(* IEC 61131-3 sources: POMIRTS_lab3/AS/Library_2/AsNxPnS, 3 files *)

(* ---- AsNxPnS.typ ---- *)
TYPE
	PnSoftwareRevisionType : 	STRUCT
		Prefix : USINT;
		X : USINT;
		Y : USINT;
		Z : USINT;
	END_STRUCT;
	PnIm0Type : 	STRUCT
		VendorID : UINT;
		OrderID : ARRAY[0..19]OF USINT;
		SerialNumber : ARRAY[0..15]OF USINT;
		HardwareRevision : UINT;
		SoftwareRevision : PnSoftwareRevisionType;
		RevisionCounter : UINT;
		ProfileID : UINT;
		ProfileSpecificType : UINT;
		IMVersion : UINT;
		IMSupported : UINT;
	END_STRUCT;
	PnIm5Type : 	STRUCT
		Annotation : ARRAY[0..63]OF USINT;
		OrderID : ARRAY[0..63]OF USINT;
		VendorID : UINT;
		SerialNumber : ARRAY[0..15]OF USINT;
		HardwareRevision : UINT;
		SoftwareRevision : PnSoftwareRevisionType;
	END_STRUCT;
END_TYPE

(* ---- AsNxPnS.fun ---- *)
{REDUND_CONTEXT} {REDUND_UNREPLICABLE} FUNCTION_BLOCK nxpnsProcessAlarm		(*process alarm*)
	VAR_INPUT
		enable			: BOOL;			(*enables execution*)
		pDevice			: UDINT;		(*interface name given as a pointer, e.g., "SL<x>.SS<y>.IF<z>"*)
		deviceHandle	: UDINT;		(*profinet slave handle*)
		alarmHandle		: UDINT;		(*alarm handle*)
		userStructId	: UINT;			(*user structure identifier*)
		api				: UDINT;		(*api*)
		slot			: UDINT;		(*slot*)
		subslot			: UDINT;		(*subslot*)
		alarmDataLen	: UINT;			(*alarm data length*)
		pAlarmData		: UDINT;		(*alarm data given as pointer*)
	END_VAR
	VAR
        _state			: UINT;			(*internal variable*)
		_result			: UINT;			(*internal variable*)
        _srcId			: UDINT;		(*internal variable*)
	END_VAR
	VAR_OUTPUT
		status			: UINT;			(*execution status: ERR_OK, ERR_FUB_ENABLE_FALSE, ERR_FUB_BUSY, 0xXXXX = see help*)
		pnStatus		: UDINT;		(*profinet stack status*)
		pnIoStatus		: UDINT;		(*profinet io status*)
	END_VAR
END_FUNCTION_BLOCK

{REDUND_CONTEXT} {REDUND_UNREPLICABLE} FUNCTION_BLOCK nxpnsDiagnosisAlarm		(*diagnosis alarm*)
	VAR_INPUT
		enable			: BOOL;			(*enables execution*)
		pDevice			: UDINT;		(*interface name given as a pointer, e.g., "SL<x>.SS<y>.IF<z>"*)
		deviceHandle	: UDINT;		(*profinet slave handle*)
		alarmHandle		: UDINT;		(*alarm handle*)
		diagHandle		: UDINT;		(*diagnosis handle*)
	END_VAR
	VAR
        _state			: UINT;			(*internal variable*)
		_result			: UINT;			(*internal variable*)
        _srcId			: UDINT;		(*internal variable*)
	END_VAR
	VAR_OUTPUT
		status			: UINT;			(*execution status: ERR_OK, ERR_FUB_ENABLE_FALSE, ERR_FUB_BUSY, 0xXXXX = see help*)
		pnStatus		: UDINT;		(*profinet stack status*)
		pnIoStatus		: UDINT;		(*profinet io status*)
	END_VAR
END_FUNCTION_BLOCK

{REDUND_CONTEXT} {REDUND_UNREPLICABLE} FUNCTION_BLOCK nxpnsPlugModule			(*plug module*)
	VAR_INPUT
		enable			: BOOL;			(*enables execution*)
		pDevice			: UDINT;		(*interface name given as a pointer, e.g., "SL<x>.SS<y>.IF<z>"*)
		deviceHandle	: UDINT;		(*profinet slave handle*)
		api				: UDINT;		(*api*)
		slot			: UDINT;		(*slot*)
		moduleId		: UDINT;		(*module identifier*)
		moduleState		: UINT;			(*module state*)
	END_VAR
	VAR
        _state			: UINT;			(*internal variable*)
		_result			: UINT;			(*internal variable*)
        _srcId			: UDINT;		(*internal variable*)
	END_VAR
	VAR_OUTPUT
		status			: UINT;			(*execution status: ERR_OK, ERR_FUB_ENABLE_FALSE, ERR_FUB_BUSY, 0xXXXX = see help*)
		pnStatus		: UDINT;		(*profinet stack status*)
	END_VAR
END_FUNCTION_BLOCK

{REDUND_CONTEXT} {REDUND_UNREPLICABLE} FUNCTION_BLOCK nxpnsPullModule			(*pull module*)
	VAR_INPUT
		enable			: BOOL;			(*enables execution*)
		pDevice			: UDINT;		(*interface name given as a pointer, e.g., "SL<x>.SS<y>.IF<z>"*)
		deviceHandle	: UDINT;		(*profinet slave handle*)
		api				: UDINT;		(*api*)
		slot			: UDINT;		(*slot*)
	END_VAR
	VAR
        _state			: UINT;			(*internal variable*)
		_result			: UINT;			(*internal variable*)
        _srcId			: UDINT;		(*internal variable*)
	END_VAR
	VAR_OUTPUT
		status			: UINT;			(*execution status: ERR_OK, ERR_FUB_ENABLE_FALSE, ERR_FUB_BUSY, 0xXXXX = see help*)
		pnStatus		: UDINT;		(*profinet stack status*)
	END_VAR
END_FUNCTION_BLOCK

{REDUND_CONTEXT} {REDUND_UNREPLICABLE} FUNCTION_BLOCK nxpnsGetHandle			(*get slave handle*)
	VAR_INPUT
		enable			: BOOL;			(*enables execution*)
		pDevice			: UDINT;		(*interface name given as a pointer, e.g., "SL<x>.SS<y>.IF<z>"*)
	END_VAR
	VAR
        _state			: UINT;			(*internal variable*)
		_result			: UINT;			(*internal variable*)
        _srcId			: UDINT;		(*internal variable*)
	END_VAR
	VAR_OUTPUT
		status			: UINT;			(*execution status: ERR_OK, ERR_FUB_ENABLE_FALSE, ERR_FUB_BUSY, 0xXXXX = see help*)
		pnStatus		: UDINT;		(*profinet stack status*)
		deviceHandle	: UDINT;		(*profinet slave handle*)
	END_VAR
END_FUNCTION_BLOCK

{REDUND_CONTEXT} {REDUND_UNREPLICABLE} FUNCTION_BLOCK nxpnsAddChannelDiag		(*add channel diagnosis*)
	VAR_INPUT
		enable			: BOOL;			(*enables execution*)
		pDevice			: UDINT;		(*interface name given as a pointer, e.g., "SL<x>.SS<y>.IF<z>"*)
		api				: UDINT;		(*api*)
		slot			: UDINT;		(*slot*)
		subslot			: UDINT;		(*subslot*)
		channelNum		: UINT;			(*channel number*)
		channelProp		: UINT;			(*channel property*)
		channelErrType	: UINT;			(*channel error type*)
	END_VAR
	VAR
        _state			: UINT;			(*internal variable*)
		_result			: UINT;			(*internal variable*)
        _srcId			: UDINT;		(*internal variable*)
	END_VAR
	VAR_OUTPUT
		status			: UINT;			(*execution status: ERR_OK, ERR_FUB_ENABLE_FALSE, ERR_FUB_BUSY, 0xXXXX = see help*)
		pnStatus		: UDINT;		(*profinet stack status*)
		diagHandle		: UDINT;		(*profinet diagnosis handle*)
	END_VAR
END_FUNCTION_BLOCK

{REDUND_CONTEXT} {REDUND_UNREPLICABLE} FUNCTION_BLOCK nxpnsAddExtChannelDiag	(*add channel diagnosis*)
	VAR_INPUT
		enable			: BOOL;			(*enables execution*)
		pDevice			: UDINT;		(*interface name given as a pointer, e.g., "SL<x>.SS<y>.IF<z>"*)
		api				: UDINT;		(*api*)
		slot			: UDINT;		(*slot*)
		subslot			: UDINT;		(*subslot*)
		channelNum		: UINT;			(*channel number*)
		channelProp		: UINT;			(*channel property*)
		channelErrType	: UINT;			(*channel error type*)
		extChannelAddValue	: UDINT;	(*reserved for future use, set to zero*)
		extChannelErrType	: UINT;		(*extended channel error type*)
	END_VAR
	VAR
        _state			: UINT;			(*internal variable*)
		_result			: UINT;			(*internal variable*)
        _srcId			: UDINT;		(*internal variable*)
	END_VAR
	VAR_OUTPUT
		status			: UINT;			(*execution status: ERR_OK, ERR_FUB_ENABLE_FALSE, ERR_FUB_BUSY, 0xXXXX = see help*)
		pnStatus		: UDINT;		(*profinet stack status*)
		diagHandle		: UDINT;		(*profinet diagnosis handle*)
	END_VAR
END_FUNCTION_BLOCK

{REDUND_CONTEXT} {REDUND_UNREPLICABLE} FUNCTION_BLOCK nxpnsAddGenChannelDiag	(*add channel diagnosis*)
	VAR_INPUT
		enable			: BOOL;			(*enables execution*)
		pDevice			: UDINT;		(*interface name given as a pointer, e.g., "SL<x>.SS<y>.IF<z>"*)
		api				: UDINT;		(*api*)
		slot			: UDINT;		(*slot*)
		subslot			: UDINT;		(*subslot*)
		channelNum		: UINT;			(*channel number*)
		channelProp		: UINT;			(*channel property*)
		channelErrType	: UINT;			(*channel error type*)
		userStructId	: UINT;			(*user structure identifier*)
		diagDataLen		: UINT;			(*diagnosis data length*)
		pDiagData		: UDINT;		(*diagnosis data given as pointer*)
	END_VAR
	VAR
        _state			: UINT;			(*internal variable*)
		_result			: UINT;			(*internal variable*)
        _srcId			: UDINT;		(*internal variable*)
	END_VAR
	VAR_OUTPUT
		status			: UINT;			(*execution status: ERR_OK, ERR_FUB_ENABLE_FALSE, ERR_FUB_BUSY, 0xXXXX = see help*)
		pnStatus		: UDINT;		(*profinet stack status*)
		diagHandle		: UDINT;		(*profinet diagnosis handle*)
	END_VAR
END_FUNCTION_BLOCK

{REDUND_CONTEXT} {REDUND_UNREPLICABLE} FUNCTION_BLOCK nxpnsRemChannelDiag		(*remove channel diagnosis*)
	VAR_INPUT
		enable			: BOOL;			(*enables execution*)
		pDevice			: UDINT;		(*interface name given as a pointer, e.g., "SL<x>.SS<y>.IF<z>"*)
		diagHandle		: UDINT;		(*diagnosis handle*)
	END_VAR
	VAR
        _state			: UINT;			(*internal variable*)
		_result			: UINT;			(*internal variable*)
        _srcId			: UDINT;		(*internal variable*)
	END_VAR
	VAR_OUTPUT
		status			: UINT;			(*execution status: ERR_OK, ERR_FUB_ENABLE_FALSE, ERR_FUB_BUSY, 0xXXXX = see help*)
		pnStatus		: UDINT;		(*profinet stack status*)
	END_VAR
END_FUNCTION_BLOCK

{REDUND_CONTEXT} {REDUND_UNREPLICABLE} FUNCTION_BLOCK nxpnsSetName				(*set station name*)
	VAR_INPUT
		enable			: BOOL;			(*enables execution*)
		pDevice			: UDINT;		(*interface name given as a pointer, e.g., "SL<x>.SS<y>.IF<z>"*)
		pName			: UDINT;		(*new station name*)
	END_VAR
	VAR
        _state			: UINT;			(*internal variable*)
		_result			: UINT;			(*internal variable*)
        _srcId			: UDINT;		(*internal variable*)
	END_VAR
	VAR_OUTPUT
		status			: UINT;			(*execution status: ERR_OK, ERR_FUB_ENABLE_FALSE, ERR_FUB_BUSY, 0xXXXX = see help*)
		pnStatus		: UDINT;		(*profinet stack status*)
	END_VAR
END_FUNCTION_BLOCK

{REDUND_CONTEXT} {REDUND_UNREPLICABLE} FUNCTION_BLOCK nxpnsStartBusComm		(*start bus communication*)
	VAR_INPUT
		enable			: BOOL;			(*enables execution*)
		pDevice			: UDINT;		(*interface name given as a pointer, e.g., "SL<x>.SS<y>.IF<z>"*)
	END_VAR
	VAR
        _state			: UINT;			(*internal variable*)
		_result			: UINT;			(*internal variable*)
        _srcId			: UDINT;		(*internal variable*)
	END_VAR
	VAR_OUTPUT
		status			: UINT;			(*execution status: ERR_OK, ERR_FUB_ENABLE_FALSE, ERR_FUB_BUSY, 0xXXXX = see help*)
		pnStatus		: UDINT;		(*profinet stack status*)
	END_VAR
END_FUNCTION_BLOCK

{REDUND_CONTEXT} {REDUND_UNREPLICABLE} FUNCTION_BLOCK nxpnsGetIm0 (*Gets the I&M0 data set for this device*)
	VAR_INPUT
		enable		: BOOL;				(*Enables execution.*)
		pDevice		: UDINT;			(*Name of the profinet device e.g. SS1.IF1.*)
	END_VAR
	VAR_OUTPUT
		status		: DINT;  			(*Status information.*)
		pnStatus	: UDINT;			(*Profinet stack status*)
		IM0 		: PnIm0Type;		(*I&M0 data*)
	END_VAR
	VAR
		_state		: UINT;				(*internal variable*)
		_result		: UINT;				(*internal variable*)
        _srcId		: UDINT;			(*internal variable*)
	END_VAR
END_FUNCTION_BLOCK

{REDUND_CONTEXT} {REDUND_UNREPLICABLE} FUNCTION_BLOCK nxpnsSetOem (*Sets the OEM data for this device*)
	VAR_INPUT
		enable		: BOOL;				(*Enables execution.*)
		pDevice		: UDINT;			(*Name of the profinet device e.g. SS1.IF1.*)
		DeviceID	: UINT;				(*Profinet Device Identification*)
		DeviceType	: ARRAY[0..24]OF USINT; (*Profinet Device Type*)
		IM0 		: PnIm0Type;		(*I&M0 data to be set*)
	END_VAR
	VAR_OUTPUT
		status		: DINT;  			(*Status information.*)
		pnStatus	: UDINT;			(*Profinet stack status*)
	END_VAR
	VAR
		_state		: UINT;				(*internal variable*)
		_result		: UINT;				(*internal variable*)
        _srcId		: UDINT;			(*internal variable*)
	END_VAR
END_FUNCTION_BLOCK

{REDUND_CONTEXT} {REDUND_UNREPLICABLE} FUNCTION_BLOCK nxpnsSetIm5 (*Sets the I&M5 data for this device*)
	VAR_INPUT
		enable		: BOOL;				(*Enables execution.*)
		pDevice		: UDINT;			(*Name of the profinet device e.g. SS1.IF1.*)
		IM5 		: PnIm5Type;		(*I&M5 data to be set*)
	END_VAR
	VAR_OUTPUT
		status		: DINT;  			(*Status information.*)
		pnStatus	: UDINT;			(*Profinet stack status*)
	END_VAR
	VAR
		_state		: UINT;				(*internal variable*)
		_result		: UINT;				(*internal variable*)
        _srcId		: UDINT;			(*internal variable*)
	END_VAR
END_FUNCTION_BLOCK

(* ---- AsNxPnS.var ---- *)
VAR CONSTANT
	nxpnsERR_INVALID_DEVICE				: UINT	:= 35320;		(*error invalid device*)
	nxpnsERR_SEND_MESSAGE				: UINT	:= 35321;		(*error send message*)
	nxpnsERR_TIMEOUT					: UINT	:= 35322;		(*error timeout*)
	nxpnsERR_PROFINET_STACK				: UINT	:= 35323;		(*error receive message*)
	nxpnsERR_PARAMETER					: UINT	:= 35324;		(*error invalid parameter*)

	nxpnsMOD_PLUG_CORRECT_MOD			: UINT	:= 16#0000;		(*plug correct module*)
	nxpnsMOD_PLUG_SUBSTITUTE_MOD		: UINT	:= 16#0001;		(*plug substitute module*)

	nxpnsALARM_DATALEN_MAX				: UDINT	:= 1024;		(*max alarm data length*)

	nxpnsCERR_SHORT_CIRCUIT				: UINT	:= 16#0001;		(*channel error type short circuit*)
	nxpnsCERR_UNDERVOLTAGE				: UINT	:= 16#0002;		(*channel error type undervoltaqe*)
	nxpnsCERR_OVERVOLTAGE				: UINT	:= 16#0003;		(*channel error type overvoltage*)
	nxpnsCERR_OVERLOAD					: UINT	:= 16#0004;		(*channel error type overload*)
	nxpnsCERR_OVERTEMPERATURE			: UINT	:= 16#0005;		(*channel error type overtemperature*)
	nxpnsCERR_LINE_BREAK				: UINT	:= 16#0006;		(*channel error type line break*)
	nxpnsCERR_UPPER_LIM_VAL_EXCEEDED	: UINT	:= 16#0007;		(*channel error type upper limit value exceededd*)
	nxpnsCERR_LOWER_LIM_VAL_EXCEEDED	: UINT	:= 16#0008;		(*channel error type lower limit value exceededd*)
	nxpnsCERR_ERROR						: UINT	:= 16#0009;		(*channel error type error*)
	nxpnsCERR_SIMULATION_ACTIVE			: UINT	:= 16#000A;		(*channel error type simulation active*)
	nxpnsCERR_DATA_TRANS_IMPOSSIBLE		: UINT	:= 16#8000;		(*channel error type data transmission impossible*)
	nxpnsCERR_REMOTE_MISM				: UINT	:= 16#8001;		(*channel error type remote mismatch*)
	nxpnsCERR_MEDIA_REDUNDANCY_MIS		: UINT	:= 16#8002;		(*channel error type media redundancy mismatch*)
	nxpnsCERR_SYNC_MISMATCH				: UINT	:= 16#8003;		(*channel error type sync mismatch*)
	nxpnsCERR_ISOCHRONOUS_MODE_MIS		: UINT	:= 16#8004;		(*channel error type isochronous mode mismatch*)
	nxpnsCERR_MULTICAST_CR_MIS			: UINT	:= 16#8005;		(*channel error type multicast cr mismatch*)
	nxpnsCERR_FIBER_OPTIC_MIS			: UINT	:= 16#8007;		(*channel error type fiber optic mismatch*)
	nxpnsCERR_NET_COMP_FUNC_MIS			: UINT	:= 16#8008;		(*channel error type network component function mismatch*)
	nxpnsCERR_TIME_MIS					: UINT	:= 16#8009;		(*channel error type time mismatch*)

	nxpnsCPROP_DIAGNOSIS				: UINT	:= 16#0000;		(*channel property diagnosis*)
	nxpnsCPROP_MAINTENANCE_REQUIRED		: UINT	:= 16#0200;		(*channel property maintenance required*)
	nxpnsCPROP_MAINTENANCE_DEMANDED		: UINT	:= 16#0400;		(*channel property maintenance demanded*)
	nxpnsCPROP_QUALIFIED_DIAGNOSIS		: UINT	:= 16#0600;		(*channel property qualified diagnosis*)
END_VAR
